Staubli VAL3: start.pgx

program start()
begin
  putln("test affichage")



end
